TYPE LoggerInfluxDb :
STRUCT
	MesAlarmCode		: WORD;				// Alarm Code
END_STRUCT
END_TYPE

(* stored: Version 1.1.0.1, ProductVersion 3.1.4024.6
   DUT LoggerInfluxDb: Id {1a4d60a1-e875-4fea-b3c0-0d9000d5332b} *)
